// Mitsubishi GX Works2 project: ZP_funtion_EX5   PLC: Q03UDV

PROGRAM MAIN
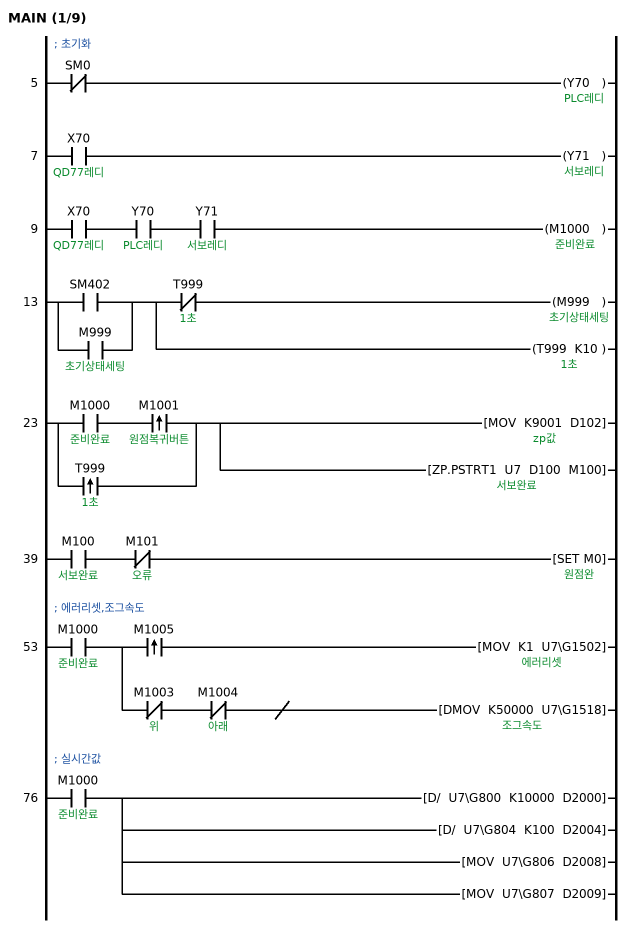
; 초기화
5     LDI     SM0
      OUT     Y70  ; PLC레디
7     LD      X70  ; QD77레디
      OUT     Y71  ; 서보레디
9     LD      X70  ; QD77레디
      AND     Y70  ; PLC레디
      AND     Y71  ; 서보레디
      OUT     M1000  ; 준비완료
13    LD      SM402
      OR      M999  ; 초기상태세팅
      MPS
      ANI     T999  ; 1초
      OUT     M999  ; 초기상태세팅
      MPP
      OUT     T999 K10  ; 1초
23    LD      M1000  ; 준비완료
      ANDP    M1001  ; 원점복귀버튼
      ORP     T999  ; 1초
      MOV     K9001 D102  ; zp값
      ZP.PSTRT1 U7 D100 M100  ; 서보완료
39    LD      M100  ; 서보완료
      ANI     M101  ; 오류
      SET     M0  ; 원점완
; 에러리셋,조그속도
53    LD      M1000  ; 준비완료
      MPS
      ANDP    M1005
      MOV     K1 U7\G1502  ; 에러리셋
      MPP
      ANI     M1003  ; 위
      ANI     M1004  ; 아래
      INV
      DMOV    K50000 U7\G1518  ; 조그속도
; 실시간값
76    LD      M1000  ; 준비완료
      D/      U7\G800 K10000 D2000
      D/      U7\G804 K100 D2004
      MOV     U7\G806 D2008
      MOV     U7\G807 D2009
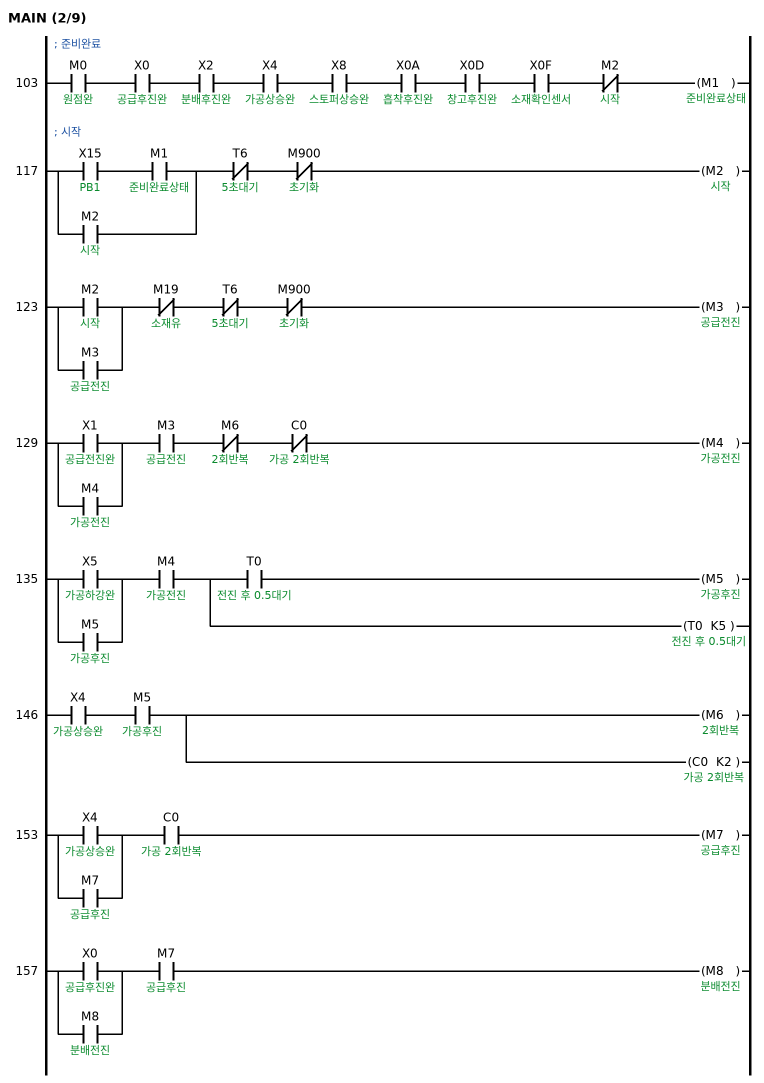
; 준비완료
103   LD      M0  ; 원점완
      AND     X0  ; 공급후진완
      AND     X2  ; 분배후진완
      AND     X4  ; 가공상승완
      AND     X8  ; 스토퍼상승완
      AND     X0A  ; 흡착후진완
      AND     X0D  ; 창고후진완
      AND     X0F  ; 소재확인센서
      ANI     M2  ; 시작
      OUT     M1  ; 준비완료상태
; 시작
117   LD      X15  ; PB1
      AND     M1  ; 준비완료상태
      OR      M2  ; 시작
      ANI     T6  ; 5초대기
      ANI     M900  ; 초기화
      OUT     M2  ; 시작
123   LD      M2  ; 시작
      OR      M3  ; 공급전진
      ANI     M19  ; 소재유
      ANI     T6  ; 5초대기
      ANI     M900  ; 초기화
      OUT     M3  ; 공급전진
129   LD      X1  ; 공급전진완
      OR      M4  ; 가공전진
      AND     M3  ; 공급전진
      ANI     M6  ; 2회반복
      ANI     C0  ; 가공 2회반복
      OUT     M4  ; 가공전진
135   LD      X5  ; 가공하강완
      OR      M5  ; 가공후진
      AND     M4  ; 가공전진
      MPS
      AND     T0  ; 전진 후 0.5대기
      OUT     M5  ; 가공후진
      MPP
      OUT     T0 K5  ; 전진 후 0.5대기
146   LD      X4  ; 가공상승완
      AND     M5  ; 가공후진
      OUT     M6  ; 2회반복
      OUT     C0 K2  ; 가공 2회반복
153   LD      X4  ; 가공상승완
      OR      M7  ; 공급후진
      AND     C0  ; 가공 2회반복
      OUT     M7  ; 공급후진
157   LD      X0  ; 공급후진완
      OR      M8  ; 분배전진
      AND     M7  ; 공급후진
      OUT     M8  ; 분배전진
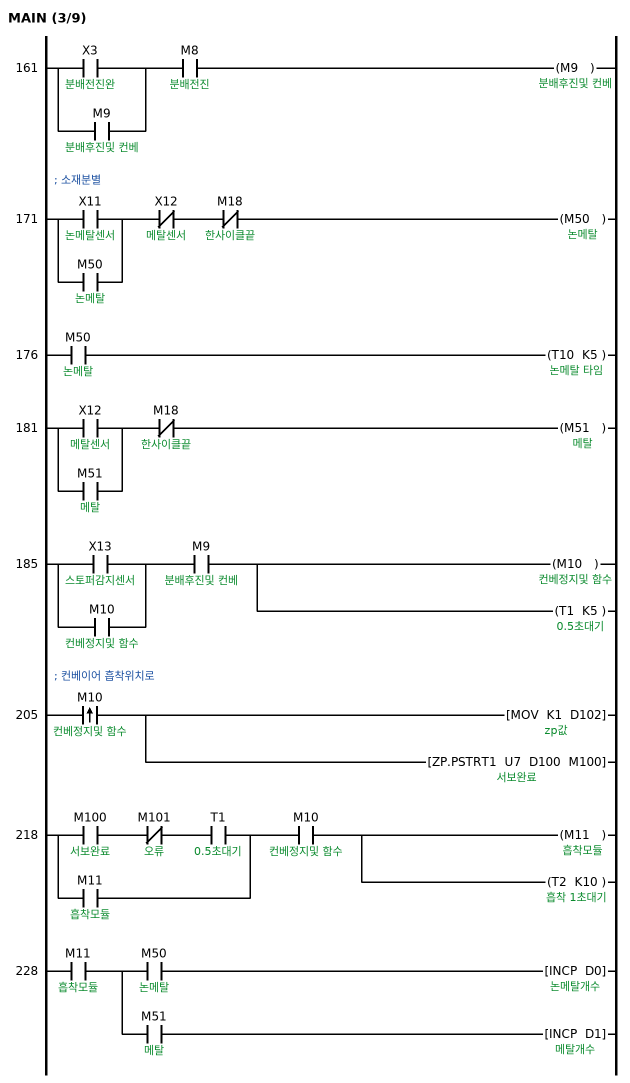
161   LD      X3  ; 분배전진완
      OR      M9  ; 분배후진및 컨베
      AND     M8  ; 분배전진
      OUT     M9  ; 분배후진및 컨베
; 소재분별
171   LD      X11  ; 논메탈센서
      OR      M50  ; 논메탈
      ANI     X12  ; 메탈센서
      ANI     M18  ; 한사이클끝
      OUT     M50  ; 논메탈
176   LD      M50  ; 논메탈
      OUT     T10 K5  ; 논메탈 타임
181   LD      X12  ; 메탈센서
      OR      M51  ; 메탈
      ANI     M18  ; 한사이클끝
      OUT     M51  ; 메탈
185   LD      X13  ; 스토퍼감지센서
      OR      M10  ; 컨베정지및 함수
      AND     M9  ; 분배후진및 컨베
      OUT     M10  ; 컨베정지및 함수
      OUT     T1 K5  ; 0.5초대기
; 컨베이어 흡착위치로
205   LDP     M10  ; 컨베정지및 함수
      MOV     K1 D102
      ZP.PSTRT1 U7 D100 M100
218   LD      M100  ; 서보완료
      ANI     M101  ; 오류
      AND     T1  ; 0.5초대기
      OR      M11  ; 흡착모듈
      AND     M10  ; 컨베정지및 함수
      OUT     M11  ; 흡착모듈
      OUT     T2 K10  ; 흡착 1초대기
228   LD      M11  ; 흡착모듈
      MPS
      AND     M50  ; 논메탈
      INCP    D0  ; 논메탈개수
      MPP
      AND     M51  ; 메탈
      INCP    D1  ; 메탈개수
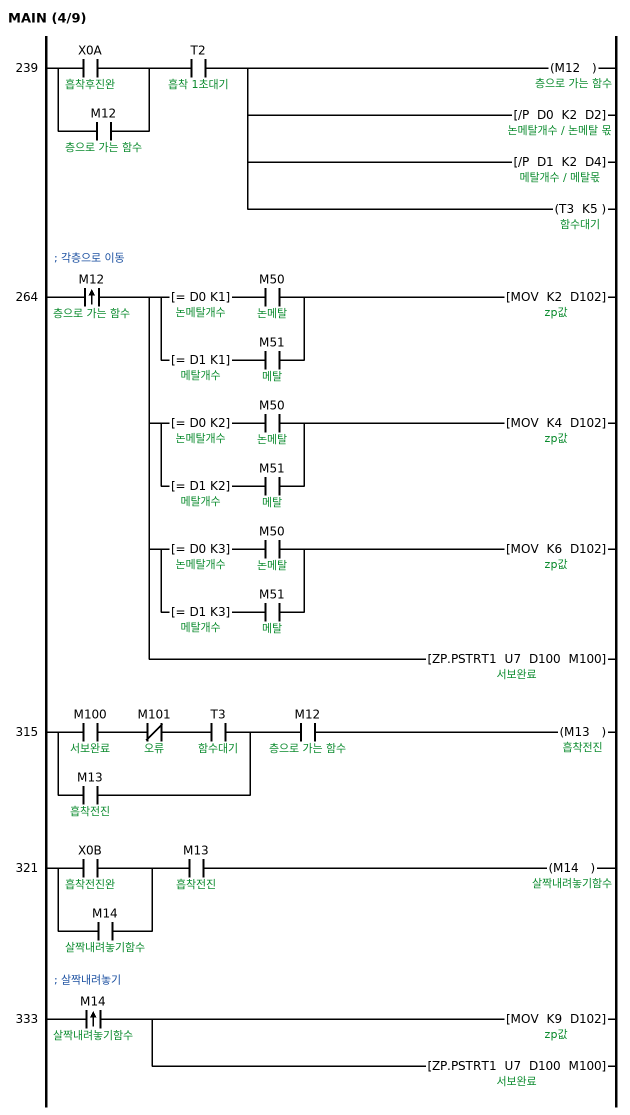
239   LD      X0A  ; 흡착후진완
      OR      M12  ; 층으로 가는 함수
      AND     T2  ; 흡착 1초대기
      OUT     M12  ; 층으로 가는 함수
      /P      D0 K2 D2  ; 논메탈 몫
      /P      D1 K2 D4  ; 메탈몫
      OUT     T3 K5  ; 함수대기
; 각층으로 이동
264   LDP     M12  ; 층으로 가는 함수
      MPS
      LD=     D0 K1  ; 논메탈개수
      AND     M50  ; 논메탈
      LD=     D1 K1  ; 메탈개수
      AND     M51  ; 메탈
      ORB
      ANB
      MOV     K2 D102
      MRD
      LD=     D0 K2  ; 논메탈개수
      AND     M50  ; 논메탈
      LD=     D1 K2  ; 메탈개수
      AND     M51  ; 메탈
      ORB
      ANB
      MOV     K4 D102
      MRD
      LD=     D0 K3  ; 논메탈개수
      AND     M50  ; 논메탈
      LD=     D1 K3  ; 메탈개수
      AND     M51  ; 메탈
      ORB
      ANB
      MOV     K6 D102
      MPP
      ZP.PSTRT1 U7 D100 M100
315   LD      M100  ; 서보완료
      ANI     M101  ; 오류
      AND     T3  ; 함수대기
      OR      M13  ; 흡착전진
      AND     M12  ; 층으로 가는 함수
      OUT     M13  ; 흡착전진
321   LD      X0B  ; 흡착전진완
      OR      M14  ; 살짝내려놓기함수
      AND     M13  ; 흡착전진
      OUT     M14  ; 살짝내려놓기함수
; 살짝내려놓기
333   LDP     M14  ; 살짝내려놓기함수
      MOV     K9 D102
      ZP.PSTRT1 U7 D100 M100
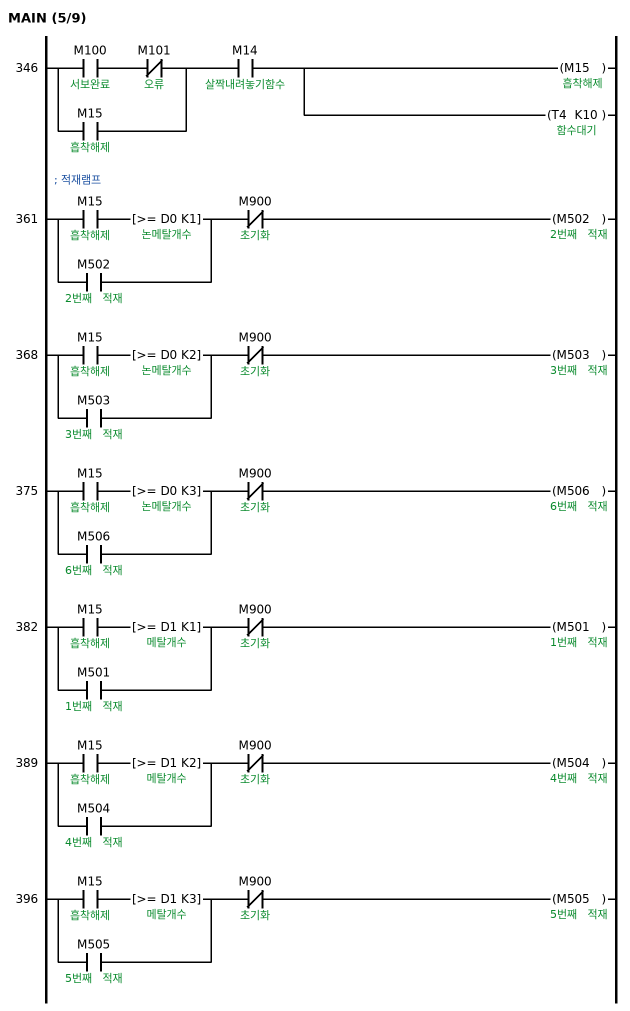
346   LD      M100  ; 서보완료
      ANI     M101  ; 오류
      OR      M15  ; 흡착해제
      AND     M14  ; 살짝내려놓기함수
      OUT     M15  ; 흡착해제
      OUT     T4 K10  ; 함수대기
; 적재램프
361   LD      M15  ; 흡착해제
      AND>=   D0 K1  ; 논메탈개수
      OR      M502  ; 2번째   적재
      ANI     M900  ; 초기화
      OUT     M502  ; 2번째   적재
368   LD      M15  ; 흡착해제
      AND>=   D0 K2  ; 논메탈개수
      OR      M503  ; 3번째   적재
      ANI     M900  ; 초기화
      OUT     M503  ; 3번째   적재
375   LD      M15  ; 흡착해제
      AND>=   D0 K3  ; 논메탈개수
      OR      M506  ; 6번째   적재
      ANI     M900  ; 초기화
      OUT     M506  ; 6번째   적재
382   LD      M15  ; 흡착해제
      AND>=   D1 K1  ; 메탈개수
      OR      M501  ; 1번째   적재
      ANI     M900  ; 초기화
      OUT     M501  ; 1번째   적재
389   LD      M15  ; 흡착해제
      AND>=   D1 K2  ; 메탈개수
      OR      M504  ; 4번째   적재
      ANI     M900  ; 초기화
      OUT     M504  ; 4번째   적재
396   LD      M15  ; 흡착해제
      AND>=   D1 K3  ; 메탈개수
      OR      M505  ; 5번째   적재
      ANI     M900  ; 초기화
      OUT     M505  ; 5번째   적재
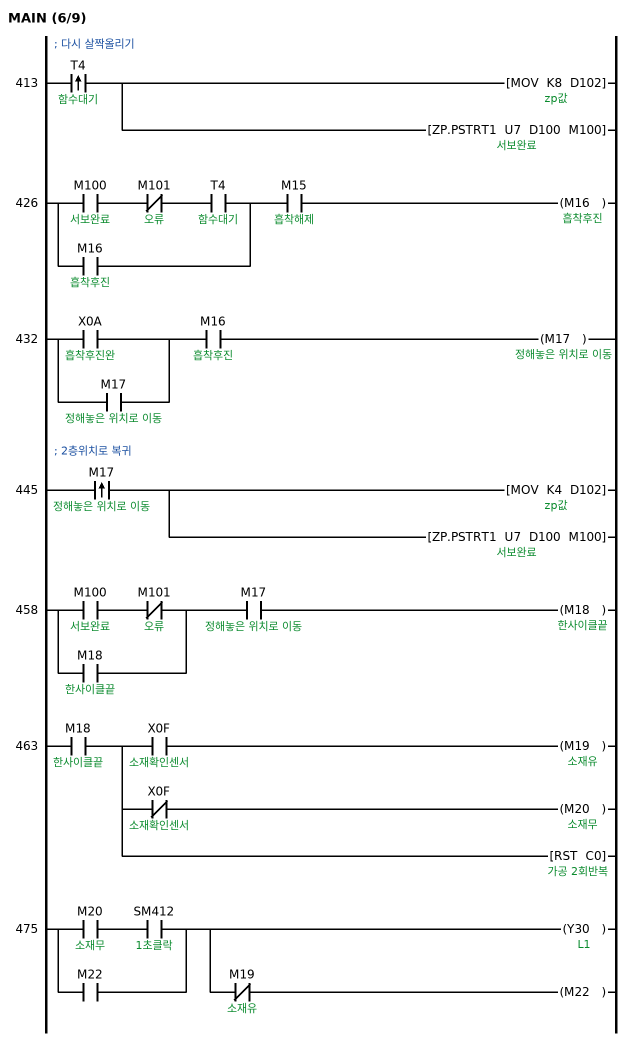
; 다시 살짝올리기
413   LDP     T4  ; 함수대기
      MOV     K8 D102
      ZP.PSTRT1 U7 D100 M100
426   LD      M100  ; 서보완료
      ANI     M101  ; 오류
      AND     T4  ; 함수대기
      OR      M16  ; 흡착후진
      AND     M15  ; 흡착해제
      OUT     M16  ; 흡착후진
432   LD      X0A  ; 흡착후진완
      OR      M17  ; 정해놓은 위치로 이동
      AND     M16  ; 흡착후진
      OUT     M17  ; 정해놓은 위치로 이동
; 2층위치로 복귀
445   LDP     M17  ; 정해놓은 위치로 이동
      MOV     K4 D102
      ZP.PSTRT1 U7 D100 M100
458   LD      M100  ; 서보완료
      ANI     M101  ; 오류
      OR      M18  ; 한사이클끝
      AND     M17  ; 정해놓은 위치로 이동
      OUT     M18  ; 한사이클끝
463   LD      M18  ; 한사이클끝
      MPS
      AND     X0F  ; 소재확인센서
      OUT     M19  ; 소재유
      MRD
      ANI     X0F  ; 소재확인센서
      OUT     M20  ; 소재무
      MPP
      RST     C0  ; 가공 2회반복
475   LD      M20  ; 소재무
      AND     SM412  ; 1초클락
      OR      M22
      OUT     Y30  ; L1
      ANI     M19  ; 소재유
      OUT     M22
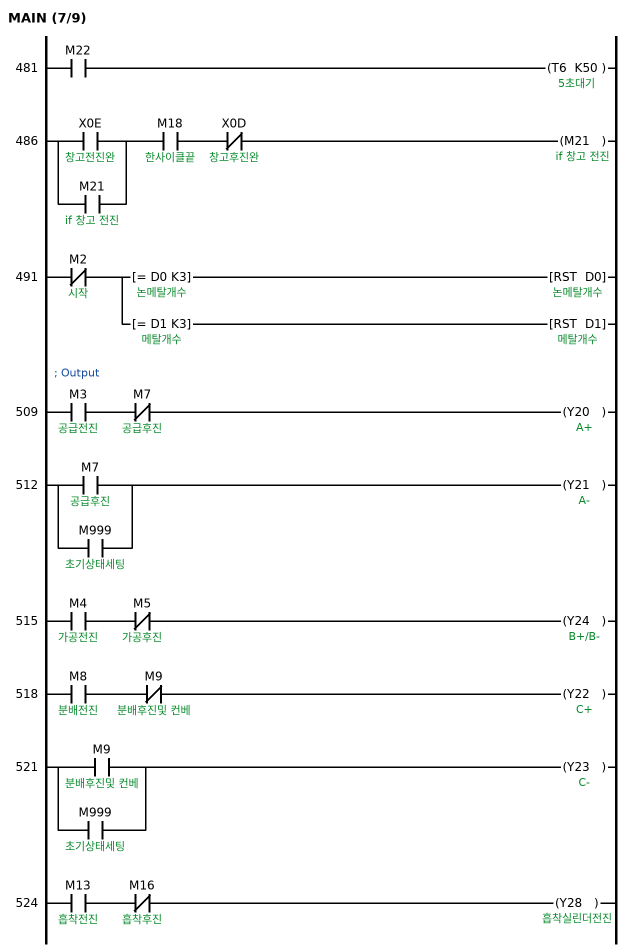
481   LD      M22
      OUT     T6 K50  ; 5초대기
486   LD      X0E  ; 창고전진완
      OR      M21  ; if 창고 전진
      AND     M18  ; 한사이클끝
      ANI     X0D  ; 창고후진완
      OUT     M21  ; if 창고 전진
491   LDI     M2  ; 시작
      MPS
      AND=    D0 K3  ; 논메탈개수
      RST     D0  ; 논메탈개수
      MPP
      AND=    D1 K3  ; 메탈개수
      RST     D1  ; 메탈개수
; Output
509   LD      M3  ; 공급전진
      ANI     M7  ; 공급후진
      OUT     Y20  ; A+
512   LD      M7  ; 공급후진
      OR      M999  ; 초기상태세팅
      OUT     Y21  ; A-
515   LD      M4  ; 가공전진
      ANI     M5  ; 가공후진
      OUT     Y24  ; B+/B-
518   LD      M8  ; 분배전진
      ANI     M9  ; 분배후진및 컨베
      OUT     Y22  ; C+
521   LD      M9  ; 분배후진및 컨베
      OR      M999  ; 초기상태세팅
      OUT     Y23  ; C-
524   LD      M13  ; 흡착전진
      ANI     M16  ; 흡착후진
      OUT     Y28  ; 흡착실린더전진
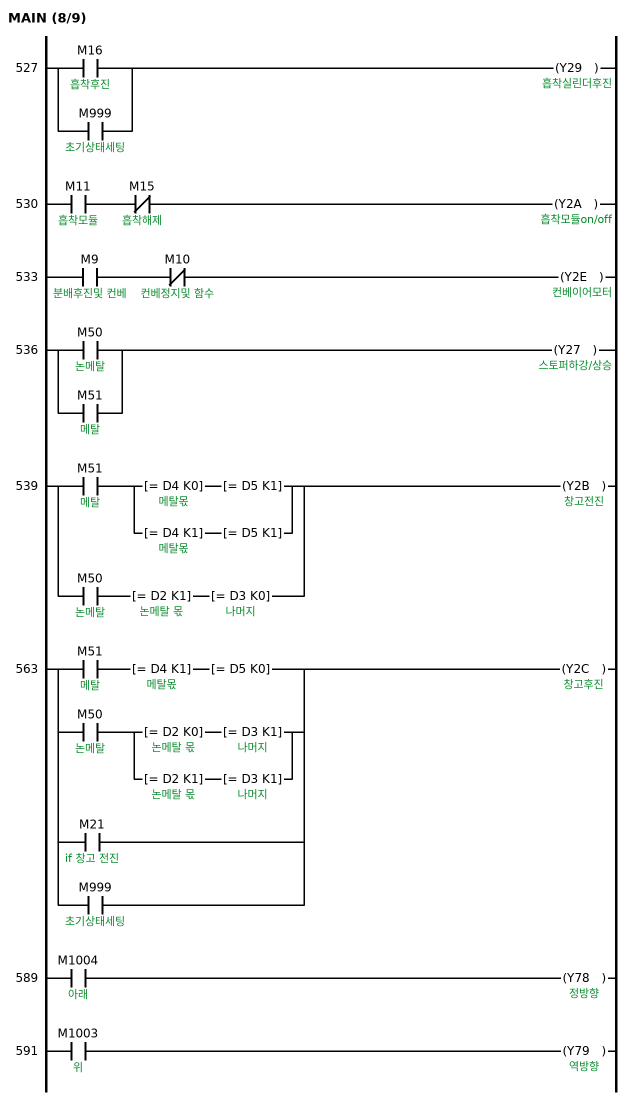
527   LD      M16  ; 흡착후진
      OR      M999  ; 초기상태세팅
      OUT     Y29  ; 흡착실린더후진
530   LD      M11  ; 흡착모듈
      ANI     M15  ; 흡착해제
      OUT     Y2A  ; 흡착모듈on/off
533   LD      M9  ; 분배후진및 컨베
      ANI     M10  ; 컨베정지및 함수
      OUT     Y2E  ; 컨베이어모터
536   LD      M50  ; 논메탈
      OR      M51  ; 메탈
      OUT     Y27  ; 스토퍼하강/상승
539   LD      M51  ; 메탈
      LD=     D4 K0  ; 메탈몫
      AND=    D5 K1
      LD=     D4 K1  ; 메탈몫
      AND=    D5 K1
      ORB
      ANB
      LD      M50  ; 논메탈
      AND=    D2 K1  ; 논메탈 몫
      AND=    D3 K0  ; 나머지
      ORB
      OUT     Y2B  ; 창고전진
563   LD      M51  ; 메탈
      AND=    D4 K1  ; 메탈몫
      AND=    D5 K0
      LD      M50  ; 논메탈
      LD=     D2 K0  ; 논메탈 몫
      AND=    D3 K1  ; 나머지
      LD=     D2 K1  ; 논메탈 몫
      AND=    D3 K1  ; 나머지
      ORB
      ANB
      ORB
      OR      M21  ; if 창고 전진
      OR      M999  ; 초기상태세팅
      OUT     Y2C  ; 창고후진
589   LD      M1004  ; 아래
      OUT     Y78  ; 정방향
591   LD      M1003  ; 위
      OUT     Y79  ; 역방향
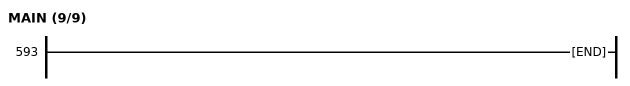
593   END
END_PROGRAM

// device comments not shown above
T5  ; 함수대기
